# EPICS substitutions: kstar/siteApp/RBA/tags/20120203-LabVIEW-version/RBAApp/Db/user.substitutions
# Example substitutions file

file "db/dbExample1.db" {
    { user = "kstar" }
}

file db/dbExample2.db {
    pattern { user, no, scan }
        { "kstar", 1, "1 second" }
        { "kstar", 2, "2 second" }
        { "kstar", 3, "5 second" }
}
